(* IEC 61131-3 sources: Structured-Text/Source Code/Logic/TRIG, 1 file *)

(* ---- Local Variables.ST ---- *)
VAR_INPUT
	IN: BOOL;
END_VAR

VAR_OUTPUT
	RTRIG_TON: BOOL;
	FTRIG_TON: BOOL;
	RTRIG_TOF: BOOL;
	FTRIG_TOF: BOOL;
END_VAR

VAR
	TON_1:			TON;
	TOF_1:			TOF;
	RISING_TON:		R_TRIG;
	FALLING_TON:	F_TRIG;
	TIME_DELAY:		TIME;
	RISING_TOF:		R_TRIG;
	FALLING_TOF:	F_TRIG;
END_VAR
